{attribute 'linkalways'} 
{attribute 'no_explicit_call' := 'This FB is a CLASS and must be accessed using methods or properties'}
{attribute 'enable_dynamic_creation'}
FUNCTION_BLOCK _ETcVnBlobCombination EXTENDS EnumDatatypeBase
VAR
	localData : ETcVnBlobCombination;
	activeData : REFERENCE TO ETcVnBlobCombination;
	enumBaseDatatype : _DINT(localData);
END_VAR

METHOD PRIVATE AddLocalEnumeration
VAR_INPUT
	Enumeration : T_MAXSTRING;
	Value : ETcVnBlobCombination;
END_VAR
AddEnumeration(Enumeration, Value);
END_METHOD

PROPERTY PUBLIC Address : PVOID
GET
Address := ADR(activeData);
END_GET
END_PROPERTY

METHOD PUBLIC ClearReference
VAR_INPUT
END_VAR
activeData REF= localData;
SetBaseDatatypeReference();
END_METHOD

METHOD PUBLIC Clone : I_Datatype
VAR
    pClone : POINTER TO _ETcVnBlobCombination;
END_VAR
pClone := __NEW(_ETcVnBlobCombination(InitialValue := Value));
Clone := pClone^;
END_METHOD

METHOD FB_init : BOOL
VAR_INPUT
	bInitRetains : BOOL; // if TRUE, the retain variables are initialized (warm start / cold start)
	bInCopyCode : BOOL;  // if TRUE, the instance afterwards gets moved into the copy code (online change)
	InitialValue : ETcVnBlobCombination;
END_VAR
localData := InitialValue;
AddBaseDatatype(enumBaseDatatype);
ClearReference();

AddLocalEnumeration('TCVN_BC_SMALLEST', ETcVnBlobCombination.TCVN_BC_SMALLEST);
AddLocalEnumeration('TCVN_BC_LARGEST', ETcVnBlobCombination.TCVN_BC_LARGEST);
AddLocalEnumeration('TCVN_BC_MIN_THRESHOLD', ETcVnBlobCombination.TCVN_BC_MIN_THRESHOLD);
AddLocalEnumeration('TCVN_BC_MAX_THRESHOLD', ETcVnBlobCombination.TCVN_BC_MAX_THRESHOLD);
AddLocalEnumeration('TCVN_BC_MEDIAN_THRESHOLD', ETcVnBlobCombination.TCVN_BC_MEDIAN_THRESHOLD);
END_METHOD

PROPERTY PUBLIC Identifier : T_MAXSTRING
GET
Identifier := 'ETcVnBlobCombination';
END_GET
END_PROPERTY

METHOD IsEnumeratorValueEqual : BOOL
VAR_INPUT
	Enumerator : I_KeyValueForwardEnumerator;
END_VAR
VAR
	storedValue : ETcVnBlobCombination;
END_VAR
IF NOT Enumerator.TryGet(storedValue) THEN
	RETURN;
END_IF

IsEnumeratorValueEqual := storedValue = activeData;
END_METHOD

METHOD PUBLIC MakeReferenceTo
VAR_INPUT
	ReferenceTarget : REFERENCE TO ETcVnBlobCombination;
END_VAR
activeData REF= ReferenceTarget;
SetBaseDatatypeReference();
END_METHOD

METHOD PROTECTED SetBaseDatatypeReference
VAR_INPUT
END_VAR
enumBaseDatatype.MakeReferenceTo(activeData);
END_METHOD

PROPERTY PUBLIC Size : UDINT
GET
Size := SIZEOF(activeData);
END_GET
END_PROPERTY

METHOD TryMakeReferenceTo : BOOL
VAR_INPUT
	Target : I_Datatype;
END_VAR
VAR
	targetAsEnum : I_EnumDatatype;
	pTargetData : POINTER TO ETcVnBlobCombination;
END_VAR
IF NOT Target.TryResolveAsEnumDatatype(targetAsEnum) THEN
	RETURN;
END_IF

IF targetAsEnum.Identifier <> Identifier THEN
	RETURN;
END_IF

pTargetData := Target.Address;
activeData REF= pTargetData^;
SetBaseDatatypeReference();
TryMakeReferenceTo := TRUE;
END_METHOD

PROPERTY PUBLIC Value : ETcVnBlobCombination
GET
Value := activeData;
END_GET
SET
activeData := Value;
END_SET
END_PROPERTY

END_FUNCTION_BLOCK

(* stored: Version 1.1.0.1
   POU _ETcVnBlobCombination: Id {eb397de0-200c-0444-1e71-1381b4a42ed0}, SpecialFunc None
   Folder Constructor: Id {398ab0f4-467c-0896-252b-9c52f56296c2}
   Folder Private: Id {c5864fc1-bf39-0c7e-35f9-49a886449c9f}
   Folder Protected: Id {6ba46316-5a26-0238-2110-255bf8cfce2b}
   Method AddLocalEnumeration: Id {f27ee67b-c9eb-03e1-2421-e1fafb64c359}
   Property Address: Id {39eb2951-7145-0f56-1d62-1a16cacba4aa}
   Get Get: Id {ea2c5b9b-a3ba-0f9d-22c8-c19e1f00ccce}
   Method ClearReference: Id {702e6def-9afc-0e65-0b12-b57d0a03510e}
   Method Clone: Id {15c57255-58d7-0faa-08a3-ebbbc56c585e}
   Method FB_init: Id {a2777ad2-5f78-03d0-249b-d2035462660d}
   Property Identifier: Id {e18c2dce-6893-00b8-0c12-610be43104e6}
   Get Get: Id {300241ca-4320-08bc-140c-5299ebb4889c}
   Method IsEnumeratorValueEqual: Id {a3ff0bea-8450-08f4-058e-7adca9ffe743}
   Method MakeReferenceTo: Id {60bc11e8-9c27-03a6-1d38-92b308dda095}
   Method SetBaseDatatypeReference: Id {bbc32874-3d81-0354-31f7-da9f5fc8f247}
   Property Size: Id {55952276-89b0-07fc-0614-c828a33db741}
   Get Get: Id {6787e0df-c35e-0055-08a4-86b16a9578f0}
   Method TryMakeReferenceTo: Id {2731b512-845e-01c9-3add-72474f14f76b}
   Property Value: Id {e83355d7-773c-080d-22c2-0d6d8a8f056c}
   Get Get: Id {4038299c-4f15-036c-3055-bdb337e6e538}
   Set Set: Id {6dd0818e-b46a-0a2d-33cf-f68ef25a597e} *)
